{attribute 'linkalways'} 
{attribute 'no_explicit_call' := 'This FB is a CLASS and must be accessed using methods or properties'}
{attribute 'enable_dynamic_creation'}
FUNCTION_BLOCK Node_ContainerType_Vector_TcVnKeyPoint EXTENDS Node
VAR
    out : _GUID;
END_VAR

METHOD PUBLIC  Clone : I_Node
VAR
	pNode : POINTER TO Node_ContainerType_Vector_TcVnKeyPoint;
END_VAR
pNode := __NEW(Node_ContainerType_Vector_TcVnKeyPoint);
Clone := pNode^;
END_METHOD

METHOD FB_init : BOOL
VAR_INPUT
	bInitRetains : BOOL; // if TRUE, the retain variables are initialized (warm start / cold start)
	bInCopyCode : BOOL;  // if TRUE, the instance afterwards gets moved into the copy code (online change)
END_VAR
AddOutput('out', out);
END_METHOD

METHOD PROTECTED OnExecute
out.Value := ContainerType_Vector_TcVnKeyPoint;
END_METHOD

END_FUNCTION_BLOCK

(* stored: Version 1.1.0.1, ProductVersion 3.1.4026.17
   POU Node_ContainerType_Vector_TcVnKeyPoint: Id {9c9cd11f-24ac-06f7-2eec-765bb8b480b8}, SpecialFunc None
   Folder Constructor: Id {3fed50b3-5d9b-0e71-19cf-5006932c04c0}
   Method Clone: Id {2c286597-10cc-054c-3cc6-34edc984bfd7}
   Method FB_init: Id {86a92cf1-ea98-0295-0a1f-9afaa73166cf}
   Method OnExecute: Id {9cd30122-e18c-0307-2a4a-88fd8743a935} *)
